{attribute 'qualified_only'}
{attribute 'strict'}
TYPE E_Command :
(
	Quit := 16#02,
	ChangeTag := 16#04,
	Reset := 16#16,
	SetMultiplexedMode := 16#9B,
	SetTriggerMode := 16#9C,
	SingleReadFixCode := 16#01,
	EnchancedReadFixCode := 16#1D,
	SingleReadWords := 16#10,
	EnchancedReadWords := 16#19,
	SingleWriteWords := 16#40,
	SingleWriteFixCode := 16#1F
)BYTE := Quit;
END_TYPE
//  Quit = '16#02'
//  ChangeTag = '16#04'
//  Reset = '16#16'
//  SetMultiplexedMode = '16#9B'
//  SetTriggerMode = '16#9C'
//  SingleReadFixCode = '16#01'
//  EnchancedReadFixCode = '16#1D'
//  SingleReadWords = '16#10'
//  EnchancedReadWords = '16#19'
//  SingleWriteWords = '16#40'
//  SingleWriteFixCode = '16#1F'

(* stored: Version 1.1.0.1, ProductVersion 3.1.4024.11
   EnumerationTextList E_Command: Id {33ccd2b1-a775-4831-b2cb-dd18a3fb09e3} *)
